(* Logix 5000 project; controller cal1615 1756-L62 rev 20.11; software revision 20.05; part 18 of 82 *)
(* tags used below, declared in another part *)
   FAULT : BOOL;   // Fault AFI
   HMI : BOOL;   // AFI HMI
   p01r09_pb_global_reset : BOOL;   // System Modes PB: Global Fault Reset
   p11_ai_exh_amps : REAL;   // Zone 1 Analog Input Exhaust Fan Amps
   p11_ai_exh_hz : REAL;   // Zone 1 Analog Input Exhaust Fan HZ
   p11_ai_exh_pct : REAL;   // Zone 1 Analog Input Exhaust Fan PCT
   p11_ai_exh_rpm : REAL;   // Zone 1 Analog Input Exhaust Fan RPM
   p11_ai_lfl : REAL;   // Zone 1 Analog Input Lower Flash Limit
   p11_ai_prs : REAL;   // Zone 1 Analog Input Pressure
   p11_ai_recirc_amps : REAL;   // Zone 1 Analog Input Recirc Fan Amps
   p11_ai_recirc_hz : REAL;   // Zone 1 Analog Input Supply Fan HZ
   p11_ai_recirc_pct : REAL;   // Zone 1 Analog Input Recirc Fan PCT
   p11_ai_recirc_rpm : REAL;   // Zone 1 Analog Input Recirc Fan RPM
   p11_ai_tc01 : REAL;   // Zone 1 Analog Input Control Thermocouple 1
   p11_ai_tc02 : REAL;   // Zone 1 Analog Input Control Thermocouple 2
   p11_ao_cv : REAL;   // Zone 1 Analog Output Control Valve
   p11_ao_exhaust_selected_speed : REAL;   // Zone 1 Analog Output Exhaust Fan VFD Selected Speed
   p11_ao_recirc_selected_speed : REAL;   // Zone 1 Analog Output Recirc Fan VFD Selected Speed
   p11_di_burner_auto : BOOL;   // Zone 1 Digital Input Burner Auto
   p11_di_burner_safeties_ok : BOOL;   // Zone 1 Digital Input Burner Safeties Ok
   p11_di_door_open : BOOL;   // Zone 1 Digital Input Access Door Open
   p11_di_exh : acs800_di_normal;   // Zone 1 Digital Inputs Exhaust Fan
   p11_di_exh_fan_mtr_ts : BOOL;   // Zone 1 Digital Input Exhaust Fan Motor Thermostat OK
   p11_di_exh_flow_ok : BOOL;   // Zone 1 Digital Input Exhaust Flow OK
   p11_di_flame_failure : BOOL;   // Zone 1 Digital Input Flame Failure
   p11_di_flame_on : BOOL;   // Zone 1 Digital Input Burner is On
   p11_di_fresh_air_clean : BOOL;   // Zone 1 Digital Input Fresh Air Filter Dirty
   p11_di_high_limit_temp_ok : BOOL;   // Zone 1 Digital Input High Limit Temperature OK
   p11_di_recirc : acs800_di_normal;   // Zone 1 Digital Inputs Recirc Fan
   p11_di_recirc_fan_mtr_ts : BOOL;   // Zone 1 Digital Input Recirc Fan Motor Thermostat OK
   p11_di_recirc_flow_ok : BOOL;   // Zone 1 Digital Input Recirc Flow OK
   p11_di_sp0 : BOOL;   // Zone 1 Digital Input Combustion Blower Pressure OK
   p11_di_sp00 : BOOL;   // Zone 1 Digital Input Recirculation Air Filter Dirty
   p11_di_tc01_bo : BOOL;   // Zone 1 Digital Input Control Thermocouple 1 Failure
   p11_di_tc02_bo : BOOL;   // Zone 1 Digital Input Control Thermocouple 2 Failure
   p11_di_zone_air_clean : BOOL;   // Zone 1 Digital Input Combustion Air Filter Dirty
   p11_dint_to_hmi : DINT[16];   // Zone 1 Temperature Control VFDs On
   p11_param_fast_to_soak : REAL;   // Zone 1 Parameter Fast to Soak Control
   p11_param_lfl_hhl : REAL;   // Zone 1 Parameter High High Lower Flash Limit
   p11_param_lfl_hl : REAL;   // Zone 1 Parameter High LFL Limit
   p11_param_pid1_ff : REAL;   // Zone 1 Parameter Fast PID Bias
   p11_param_pid1_kd : REAL;   // Zone 1 Parameter Fast PID Derivative Gain
   p11_param_pid1_ki : REAL;   // Zone 1 Parameter Fast PID Integral Gain
   p11_param_pid1_kp : REAL;   // Zone 1 Parameter Fast PID Proportional Gain
   p11_param_pid2_ff : REAL;   // Zone 1 Parameter Auto PID Bias
   p11_param_pid2_kd : REAL;   // Zone 1 Parameter Auto PID Derivative Gain
   p11_param_pid2_ki : REAL;   // Zone 1 Parameter Auto PID Integral Gain
   p11_param_pid2_kp : REAL;   // Zone 1 Parameter Auto PID Proportional Gain
   p11_param_shutdown_temp : REAL;   // Zone 1 Parameter Zone Shutdown Temperature
   p11_param_soak_to_fast : REAL;   // Zone 1 Parameter Soak to Fast Control
   p11_param_tc01_dev : REAL;   // Zone 1 Parameter Oven Temperature Deviation from Setpoint
   p11_param_tc01_hl : REAL;   // Zone 1 Parameter Process Air High Limit
   p11_param_tc01z : REAL;   // Zone 1 Parameter Process Temperature Zero Offset
   p11_param_tc02z : REAL;   // Zone 1 Parameter SupplyTemperature Zero Offset
   p11_param_zone_pressure : REAL;   // Zone 1 Parameter High Pressure LImit
   p11_real_to_hmi : REAL[112];   // Zone 1 Real to HMI
   p11r01 : routine;   // Zone 1 Main
   p11r05 : routine;   // Zone 1 Dint to HMI
   p11r05_exh_status : DINT;
   p11r05_recirc_status : DINT;
   p11r05_temp_ctrl_status : DINT;
   p11r05_timer_fault : TIMER[4];   // Zone 1 Dint to HMI Fault Delay
   p11r05_timer_warning : TIMER[4];   // Zone 1 Dint to HMI Warning Delay
   p11r06 : routine;   // Zone 1 Real to HMI
   p11r06_timer_fault : TIMER[4];   // Zone 1 Real to HMI Fault Delay
   p11r06_timer_warning : TIMER[4];   // Zone 1 Real to HMI Warning Delay
   p11r20_state : DINT;   // Zone 1 Temperature Control State
   p11r20_status : DINT;   // Zone 1 Temperature Control Sequence Status
   p11r30 : routine;   // Zone 1 Temperature Control
   p11r30_cv_man_sp : REAL;   // Zone 1 Temperature Control Manual Heat Control Valve Setpoint
   p11r30_permissive_run : BOOL;   // Zone 1 Temperature Control Run Permissive
   p11r30_pid_temp : PID;   // Zone 1 Temperature Control PID
   p11r30_pid_temp_pv : REAL;   // Zone 1 Temperature Control PID Temp Process Variable
   p11r30_pid_temp_sp : REAL;   // Zone 1 Temperature Control PID Temperature Control Setpoint
   p11r30_request_heat : BOOL;   // Zone 1 Temperature Control Request Heat
   p11r30_request_manual : BOOL;   // Zone 1 Temperature Control Request Manual Control
   p11r30_vfds_ready : BOOL;   // Zone 1 Temperature Control VFDs On
   p11r31 : routine;   // Zone 1 Exhaust VFD
   p11r31_request_auto_run : BOOL;   // Zone 1 Exhaust Fan Run Request
   p11r31_request_auto_stop : BOOL;   // Zone 1 Exhaust VFD Request Auto Stop
   p11r31_vfd_stopped : BOOL;   // Zone 1 Exhaust VFD VFD Stopped
   p11r32 : routine;   // Zone 1 Recirc VFD
   p11r32_request_auto_run : BOOL;   // Zone 1 Recirc Fan Run Request
   p11r32_request_auto_stop : BOOL;   // Zone 1 Recirc VFD Request Auto Stop
   p11r32_vfd_stopped : BOOL;   // Zone 1 Recirc VFD VFD Stopped
(* P11_Zone_1, continued *)

ROUTINE R05_Dint_to_HMI   (* ladder *)
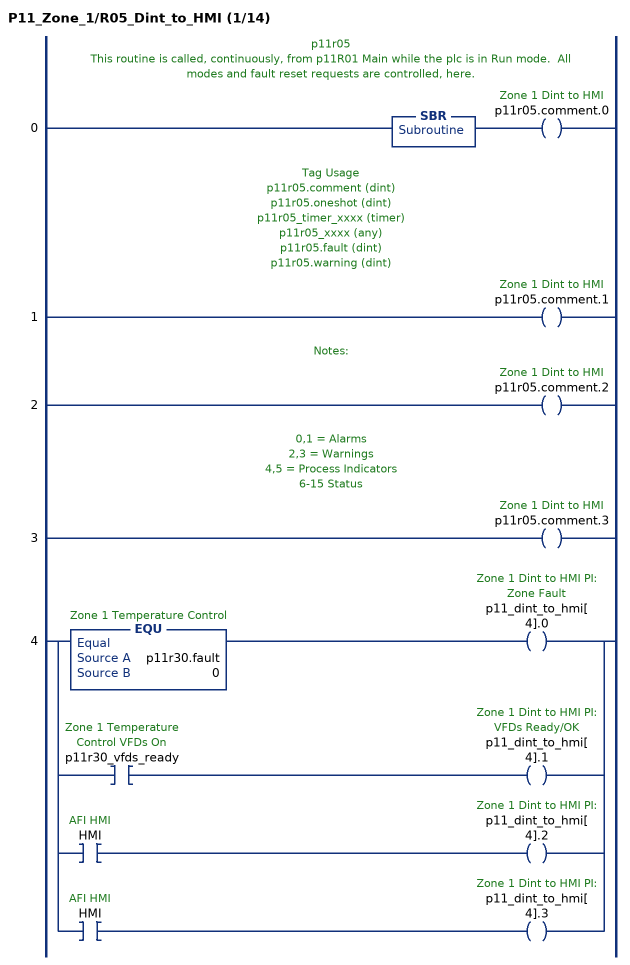
   // p11r05
   // This routine is called, continuously, from p11R01 Main while the plc is in Run mode.  All modes and fault reset requests are controlled, here.
   0: SBR()OTE(p11r05.comment.0);
   // Tag Usage
   // p11r05.comment (dint)
   // p11r05.oneshot (dint)
   // p11r05_timer_xxxx (timer)
   // p11r05_xxxx (any)
   // p11r05.fault (dint)
   // p11r05.warning (dint)
   1: OTE(p11r05.comment.1);
   // Notes:
   2: OTE(p11r05.comment.2);
   // 0,1 = Alarms
   // 2,3 = Warnings
   // 4,5 = Process Indicators
   // 6-15 Status
   3: OTE(p11r05.comment.3);
   4: [EQU(p11r30.fault,0) OTE(p11_dint_to_hmi[4].0) ,XIC(p11r30_vfds_ready) OTE(p11_dint_to_hmi[4].1) ,XIC(HMI) OTE(p11_dint_to_hmi[4].2) ,XIC(HMI) OTE(p11_dint_to_hmi[4].3) ];
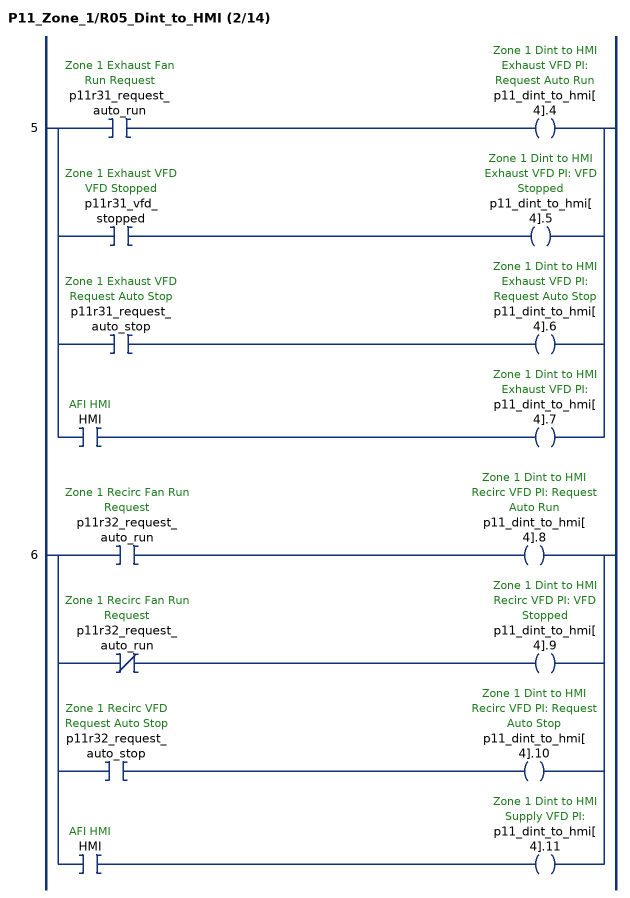
   5: [XIC(p11r31_request_auto_run) OTE(p11_dint_to_hmi[4].4) ,XIC(p11r31_vfd_stopped) OTE(p11_dint_to_hmi[4].5) ,XIC(p11r31_request_auto_stop) OTE(p11_dint_to_hmi[4].6) ,XIC(HMI) OTE(p11_dint_to_hmi[4].7) ];
   6: [XIC(p11r32_request_auto_run) OTE(p11_dint_to_hmi[4].8) ,XIO(p11r32_request_auto_run) OTE(p11_dint_to_hmi[4].9) ,XIC(p11r32_request_auto_stop) OTE(p11_dint_to_hmi[4].10) ,XIC(HMI) OTE(p11_dint_to_hmi[4].11) ];
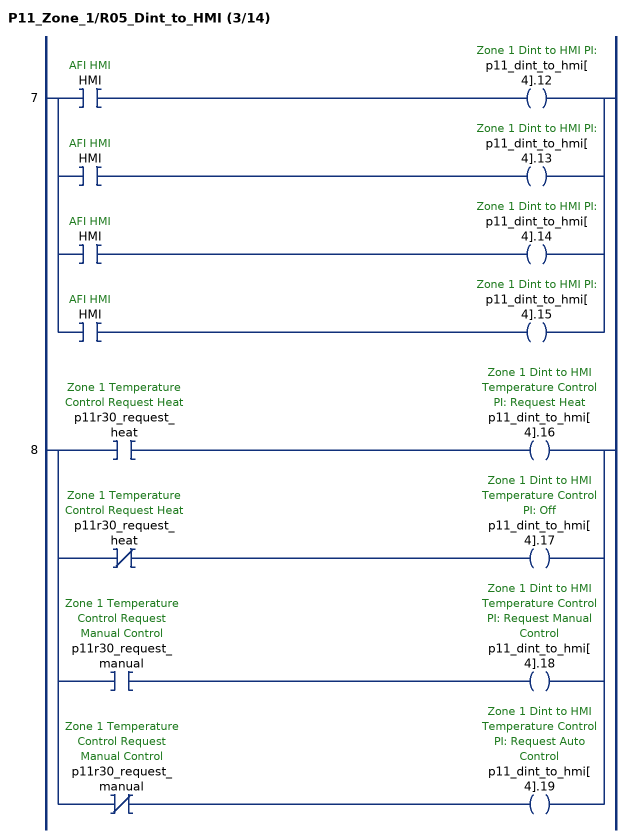
   7: [XIC(HMI) OTE(p11_dint_to_hmi[4].12) ,XIC(HMI) OTE(p11_dint_to_hmi[4].13) ,XIC(HMI) OTE(p11_dint_to_hmi[4].14) ,XIC(HMI) OTE(p11_dint_to_hmi[4].15) ];
   8: [XIC(p11r30_request_heat) OTE(p11_dint_to_hmi[4].16) ,XIO(p11r30_request_heat) OTE(p11_dint_to_hmi[4].17) ,XIC(p11r30_request_manual) OTE(p11_dint_to_hmi[4].18) ,XIO(p11r30_request_manual) OTE(p11_dint_to_hmi[4].19) ];
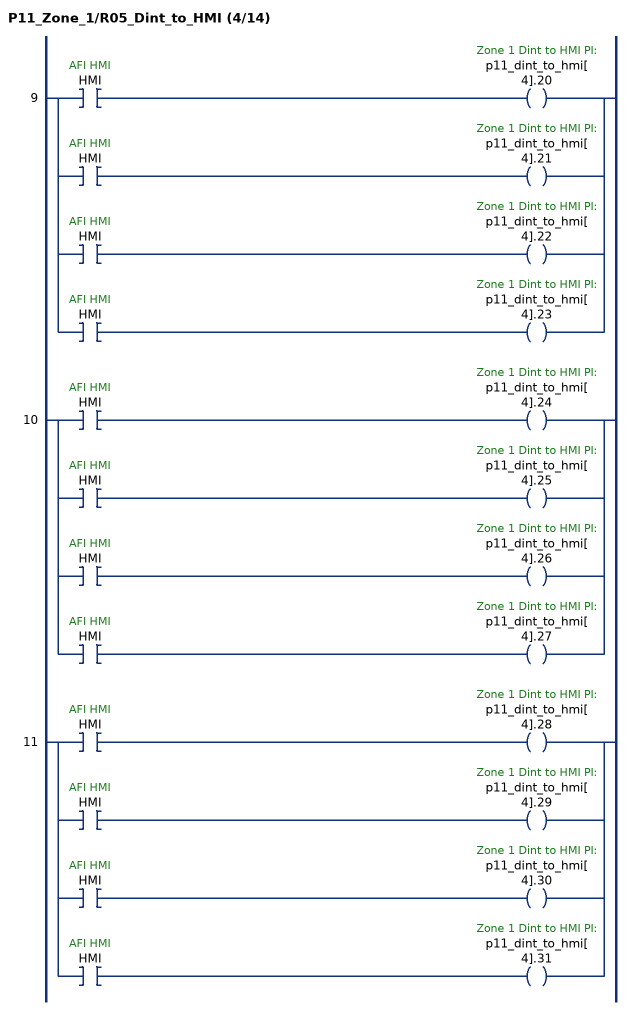
   9: [XIC(HMI) OTE(p11_dint_to_hmi[4].20) ,XIC(HMI) OTE(p11_dint_to_hmi[4].21) ,XIC(HMI) OTE(p11_dint_to_hmi[4].22) ,XIC(HMI) OTE(p11_dint_to_hmi[4].23) ];
   10: [XIC(HMI) OTE(p11_dint_to_hmi[4].24) ,XIC(HMI) OTE(p11_dint_to_hmi[4].25) ,XIC(HMI) OTE(p11_dint_to_hmi[4].26) ,XIC(HMI) OTE(p11_dint_to_hmi[4].27) ];
   11: [XIC(HMI) OTE(p11_dint_to_hmi[4].28) ,XIC(HMI) OTE(p11_dint_to_hmi[4].29) ,XIC(HMI) OTE(p11_dint_to_hmi[4].30) ,XIC(HMI) OTE(p11_dint_to_hmi[4].31) ];
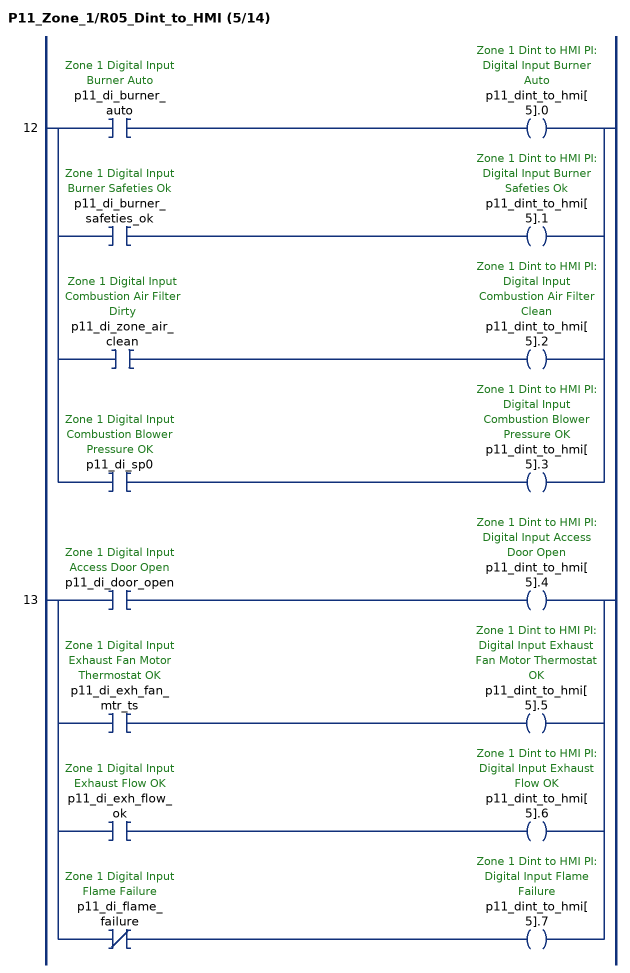
   12: [XIC(p11_di_burner_auto) OTE(p11_dint_to_hmi[5].0) ,XIC(p11_di_burner_safeties_ok) OTE(p11_dint_to_hmi[5].1) ,XIC(p11_di_zone_air_clean) OTE(p11_dint_to_hmi[5].2) ,XIC(p11_di_sp0) OTE(p11_dint_to_hmi[5].3) ];
   13: [XIC(p11_di_door_open) OTE(p11_dint_to_hmi[5].4) ,XIC(p11_di_exh_fan_mtr_ts) OTE(p11_dint_to_hmi[5].5) ,XIC(p11_di_exh_flow_ok) OTE(p11_dint_to_hmi[5].6) ,XIO(p11_di_flame_failure) OTE(p11_dint_to_hmi[5].7) ];
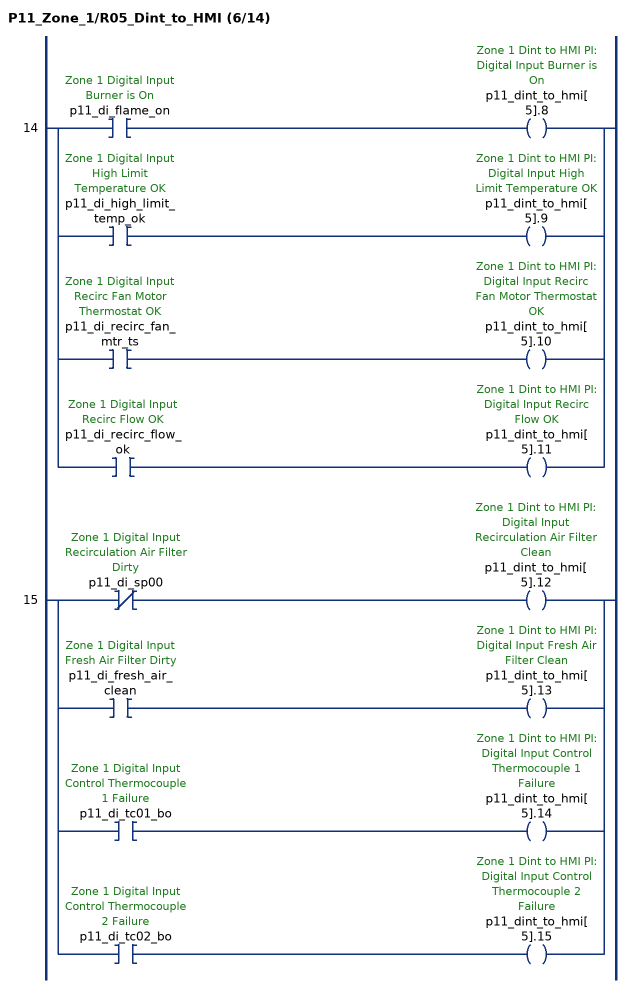
   14: [XIC(p11_di_flame_on) OTE(p11_dint_to_hmi[5].8) ,XIC(p11_di_high_limit_temp_ok) OTE(p11_dint_to_hmi[5].9) ,XIC(p11_di_recirc_fan_mtr_ts) OTE(p11_dint_to_hmi[5].10) ,XIC(p11_di_recirc_flow_ok) OTE(p11_dint_to_hmi[5].11) ];
   15: [XIO(p11_di_sp00) OTE(p11_dint_to_hmi[5].12) ,XIC(p11_di_fresh_air_clean) OTE(p11_dint_to_hmi[5].13) ,XIC(p11_di_tc01_bo) OTE(p11_dint_to_hmi[5].14) ,XIC(p11_di_tc02_bo) OTE(p11_dint_to_hmi[5].15) ];
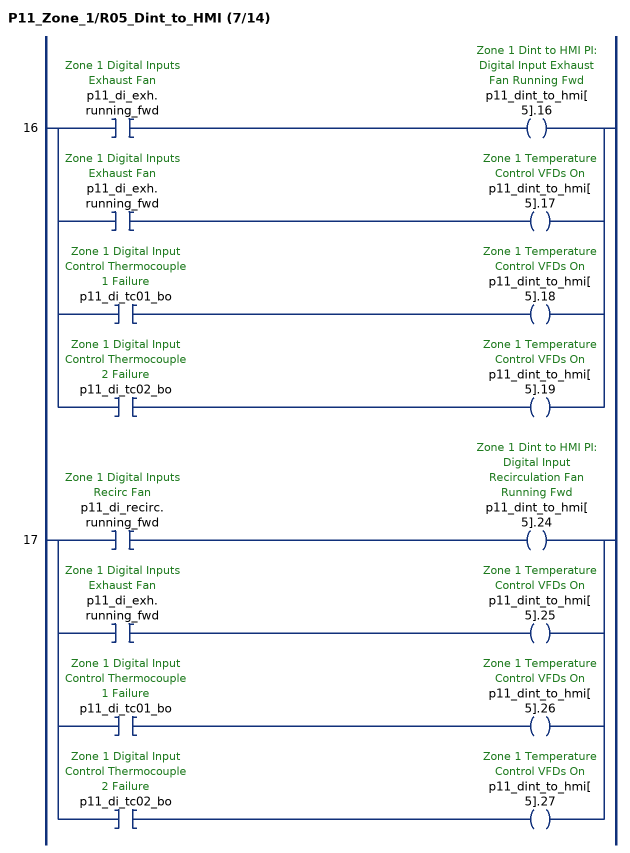
   16: [XIC(p11_di_exh.running_fwd) OTE(p11_dint_to_hmi[5].16) ,XIC(p11_di_exh.running_fwd) OTE(p11_dint_to_hmi[5].17) ,XIC(p11_di_tc01_bo) OTE(p11_dint_to_hmi[5].18) ,XIC(p11_di_tc02_bo) OTE(p11_dint_to_hmi[5].19) ];
   17: [XIC(p11_di_recirc.running_fwd) OTE(p11_dint_to_hmi[5].24) ,XIC(p11_di_exh.running_fwd) OTE(p11_dint_to_hmi[5].25) ,XIC(p11_di_tc01_bo) OTE(p11_dint_to_hmi[5].26) ,XIC(p11_di_tc02_bo) OTE(p11_dint_to_hmi[5].27) ];
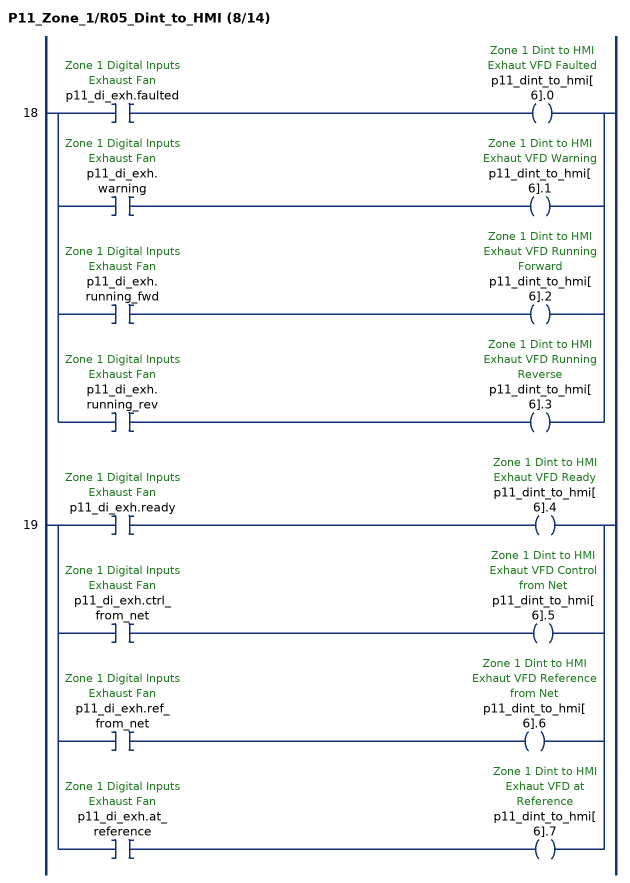
   18: [XIC(p11_di_exh.faulted) OTE(p11_dint_to_hmi[6].0) ,XIC(p11_di_exh.warning) OTE(p11_dint_to_hmi[6].1) ,XIC(p11_di_exh.running_fwd) OTE(p11_dint_to_hmi[6].2) ,XIC(p11_di_exh.running_rev) OTE(p11_dint_to_hmi[6].3) ];
   19: [XIC(p11_di_exh.ready) OTE(p11_dint_to_hmi[6].4) ,XIC(p11_di_exh.ctrl_from_net) OTE(p11_dint_to_hmi[6].5) ,XIC(p11_di_exh.ref_from_net) OTE(p11_dint_to_hmi[6].6) ,XIC(p11_di_exh.at_reference) OTE(p11_dint_to_hmi[6].7) ];
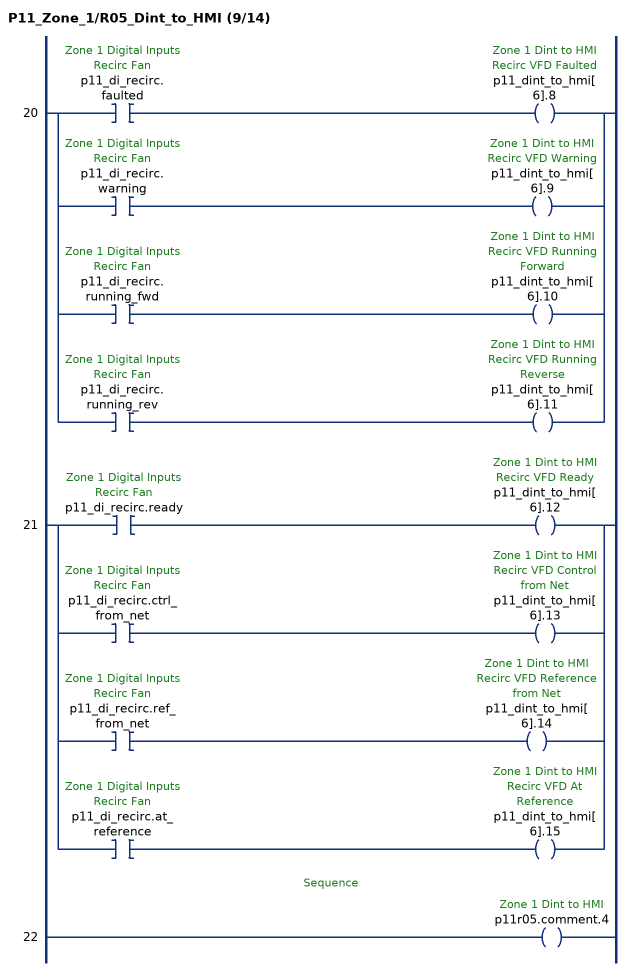
   20: [XIC(p11_di_recirc.faulted) OTE(p11_dint_to_hmi[6].8) ,XIC(p11_di_recirc.warning) OTE(p11_dint_to_hmi[6].9) ,XIC(p11_di_recirc.running_fwd) OTE(p11_dint_to_hmi[6].10) ,XIC(p11_di_recirc.running_rev) OTE(p11_dint_to_hmi[6].11) ];
   21: [XIC(p11_di_recirc.ready) OTE(p11_dint_to_hmi[6].12) ,XIC(p11_di_recirc.ctrl_from_net) OTE(p11_dint_to_hmi[6].13) ,XIC(p11_di_recirc.ref_from_net) OTE(p11_dint_to_hmi[6].14) ,XIC(p11_di_recirc.at_reference) OTE(p11_dint_to_hmi[6].15) ];
   // Sequence
   22: OTE(p11r05.comment.4);
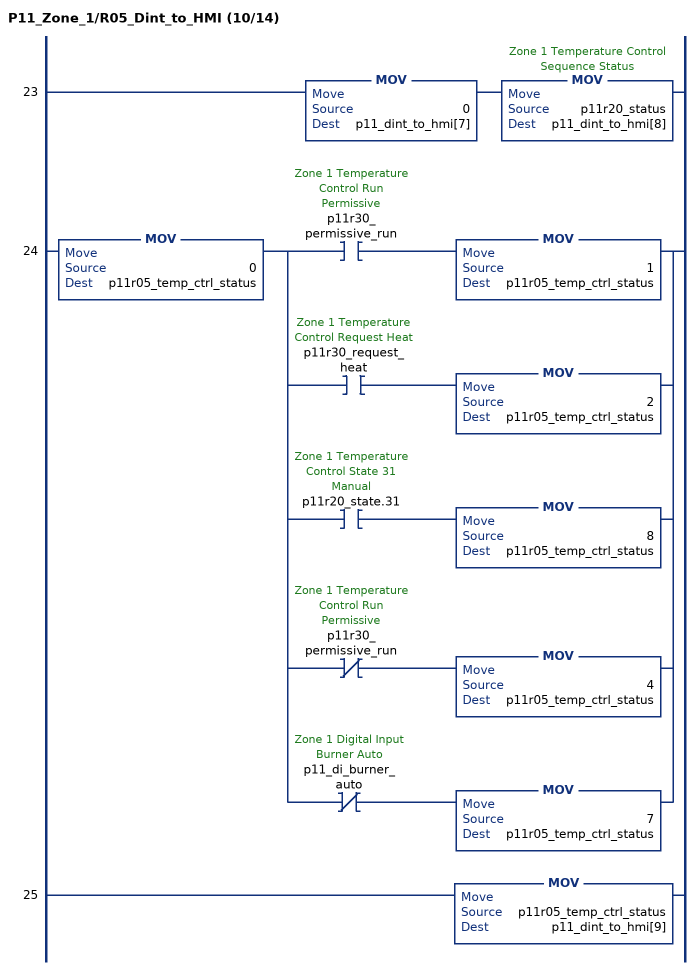
   23: MOV(0,p11_dint_to_hmi[7])MOV(p11r20_status,p11_dint_to_hmi[8]);
   24: MOV(0,p11r05_temp_ctrl_status)[XIC(p11r30_permissive_run) MOV(1,p11r05_temp_ctrl_status) ,XIC(p11r30_request_heat) MOV(2,p11r05_temp_ctrl_status) ,XIC(p11r20_state.31) MOV(8,p11r05_temp_ctrl_status) ,XIO(p11r30_permissive_run) MOV(4,p11r05_temp_ctrl_status) ,XIO(p11_di_burner_auto) MOV(7,p11r05_temp_ctrl_status) ];
   25: MOV(p11r05_temp_ctrl_status,p11_dint_to_hmi[9]);
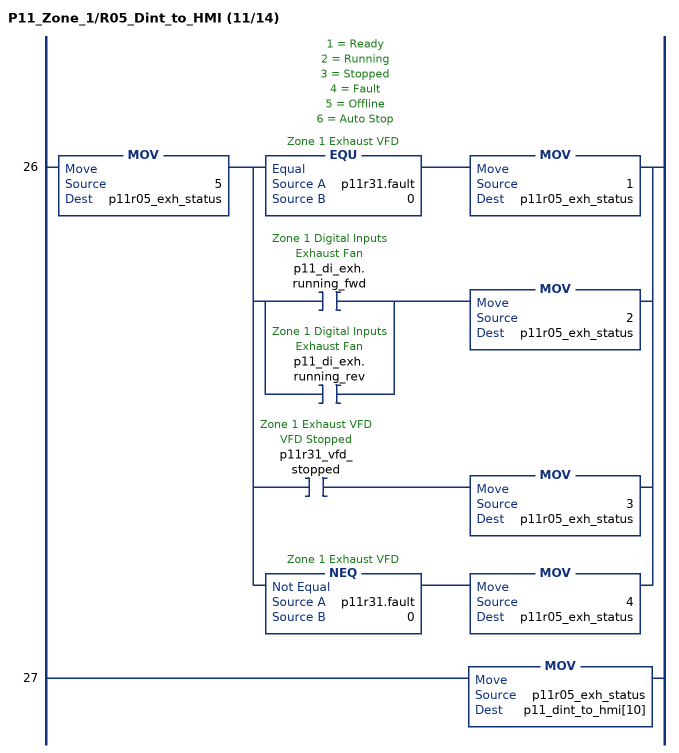
   // 1 = Ready
   // 2 = Running
   // 3 = Stopped
   // 4 = Fault
   // 5 = Offline
   // 6 = Auto Stop
   26: MOV(5,p11r05_exh_status)[EQU(p11r31.fault,0) MOV(1,p11r05_exh_status) ,[XIC(p11_di_exh.running_fwd) ,XIC(p11_di_exh.running_rev) ] MOV(2,p11r05_exh_status) ,XIC(p11r31_vfd_stopped) MOV(3,p11r05_exh_status) ,NEQ(p11r31.fault,0) MOV(4,p11r05_exh_status) ];
   27: MOV(p11r05_exh_status,p11_dint_to_hmi[10]);
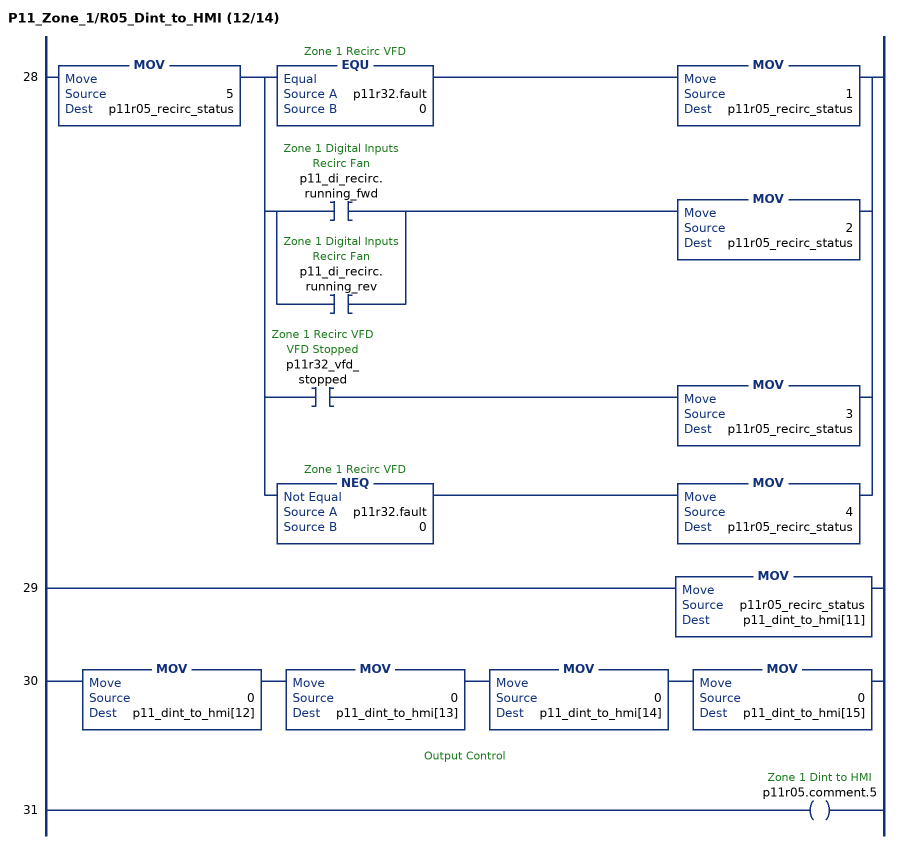
   28: MOV(5,p11r05_recirc_status)[EQU(p11r32.fault,0) MOV(1,p11r05_recirc_status) ,[XIC(p11_di_recirc.running_fwd) ,XIC(p11_di_recirc.running_rev) ] MOV(2,p11r05_recirc_status) ,XIC(p11r32_vfd_stopped) MOV(3,p11r05_recirc_status) ,NEQ(p11r32.fault,0) MOV(4,p11r05_recirc_status) ];
   29: MOV(p11r05_recirc_status,p11_dint_to_hmi[11]);
   30: MOV(0,p11_dint_to_hmi[12])MOV(0,p11_dint_to_hmi[13])MOV(0,p11_dint_to_hmi[14])MOV(0,p11_dint_to_hmi[15]);
   // Output Control
   31: OTE(p11r05.comment.5);
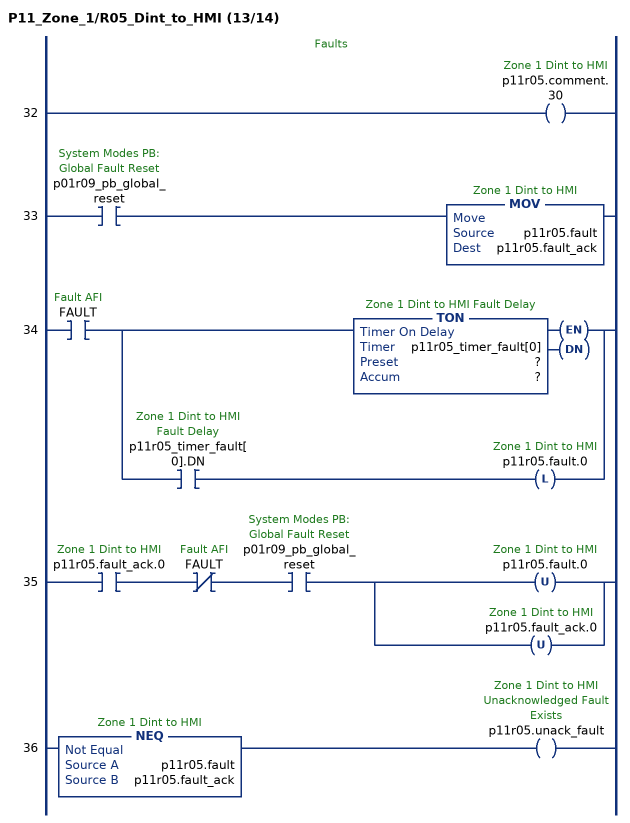
   // Faults
   32: OTE(p11r05.comment.30);
   33: XIC(p01r09_pb_global_reset)MOV(p11r05.fault,p11r05.fault_ack);
   34: XIC(FAULT)[TON(p11r05_timer_fault[0],?,?) ,XIC(p11r05_timer_fault[0].DN) OTL(p11r05.fault.0) ];
   35: XIC(p11r05.fault_ack.0)XIO(FAULT)XIC(p01r09_pb_global_reset)[OTU(p11r05.fault.0) ,OTU(p11r05.fault_ack.0) ];
   36: NEQ(p11r05.fault,p11r05.fault_ack)OTE(p11r05.unack_fault);
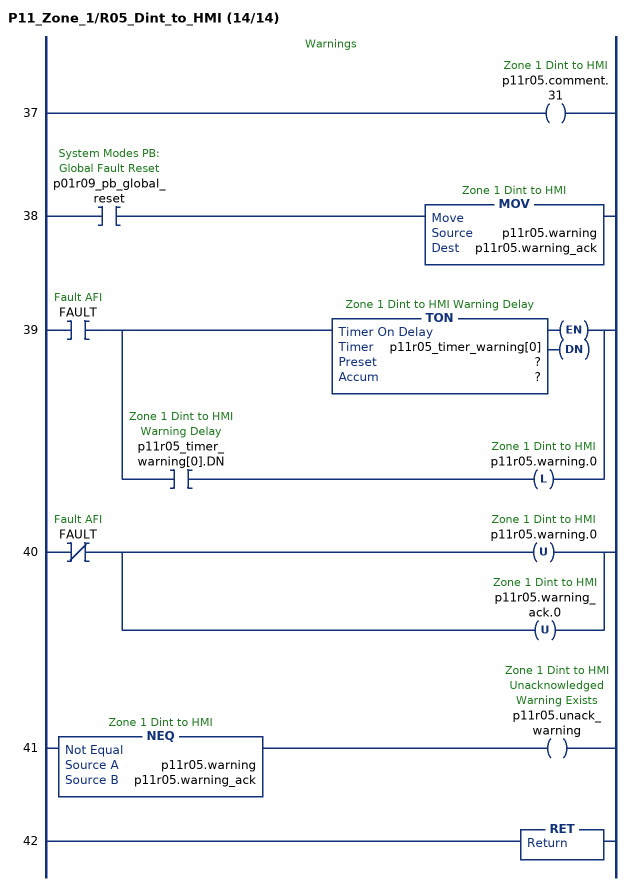
   // Warnings
   37: OTE(p11r05.comment.31);
   38: XIC(p01r09_pb_global_reset)MOV(p11r05.warning,p11r05.warning_ack);
   39: XIC(FAULT)[TON(p11r05_timer_warning[0],?,?) ,XIC(p11r05_timer_warning[0].DN) OTL(p11r05.warning.0) ];
   40: XIO(FAULT)[OTU(p11r05.warning.0) ,OTU(p11r05.warning_ack.0) ];
   41: NEQ(p11r05.warning,p11r05.warning_ack)OTE(p11r05.unack_warning);
   42: RET();
END_ROUTINE

ROUTINE R06_Real_to_HMI   (* ladder *)
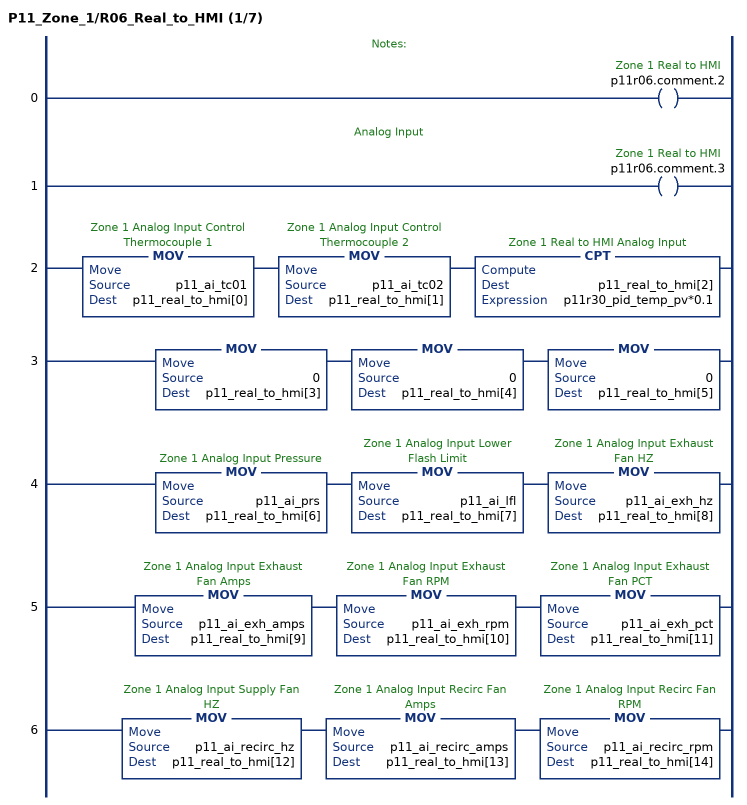
   // Notes:
   0: OTE(p11r06.comment.2);
   // Analog Input
   1: OTE(p11r06.comment.3);
   2: MOV(p11_ai_tc01,p11_real_to_hmi[0])MOV(p11_ai_tc02,p11_real_to_hmi[1])CPT(p11_real_to_hmi[2],p11r30_pid_temp_pv*0.1);
   3: MOV(0,p11_real_to_hmi[3])MOV(0,p11_real_to_hmi[4])MOV(0,p11_real_to_hmi[5]);
   4: MOV(p11_ai_prs,p11_real_to_hmi[6])MOV(p11_ai_lfl,p11_real_to_hmi[7])MOV(p11_ai_exh_hz,p11_real_to_hmi[8]);
   5: MOV(p11_ai_exh_amps,p11_real_to_hmi[9])MOV(p11_ai_exh_rpm,p11_real_to_hmi[10])MOV(p11_ai_exh_pct,p11_real_to_hmi[11]);
   6: MOV(p11_ai_recirc_hz,p11_real_to_hmi[12])MOV(p11_ai_recirc_amps,p11_real_to_hmi[13])MOV(p11_ai_recirc_rpm,p11_real_to_hmi[14]);
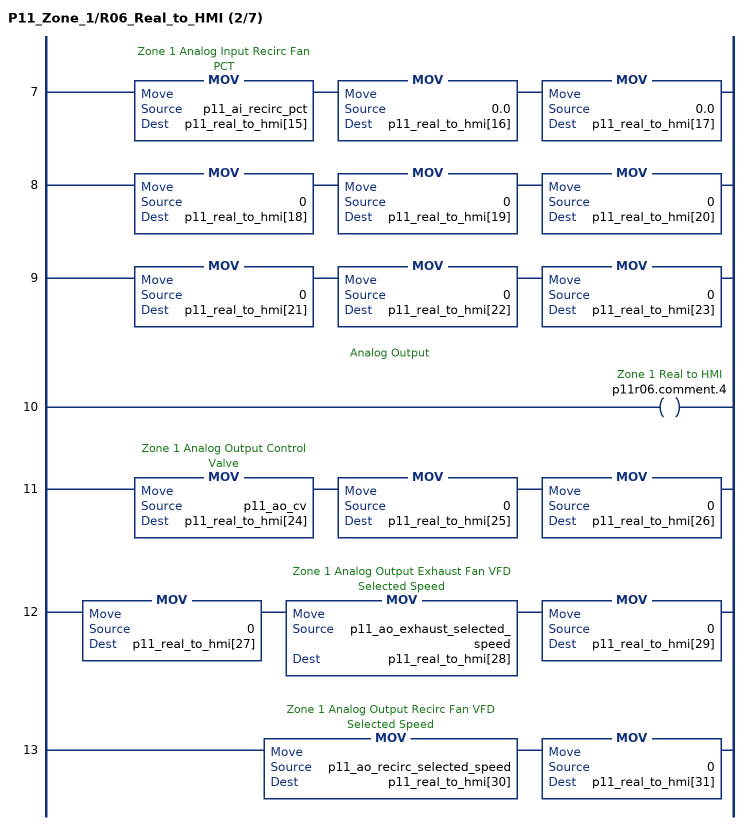
   7: MOV(p11_ai_recirc_pct,p11_real_to_hmi[15])MOV(0.0,p11_real_to_hmi[16])MOV(0.0,p11_real_to_hmi[17]);
   8: MOV(0,p11_real_to_hmi[18])MOV(0,p11_real_to_hmi[19])MOV(0,p11_real_to_hmi[20]);
   9: MOV(0,p11_real_to_hmi[21])MOV(0,p11_real_to_hmi[22])MOV(0,p11_real_to_hmi[23]);
   // Analog Output
   10: OTE(p11r06.comment.4);
   11: MOV(p11_ao_cv,p11_real_to_hmi[24])MOV(0,p11_real_to_hmi[25])MOV(0,p11_real_to_hmi[26]);
   12: MOV(0,p11_real_to_hmi[27])MOV(p11_ao_exhaust_selected_speed,p11_real_to_hmi[28])MOV(0,p11_real_to_hmi[29]);
   13: MOV(p11_ao_recirc_selected_speed,p11_real_to_hmi[30])MOV(0,p11_real_to_hmi[31]);
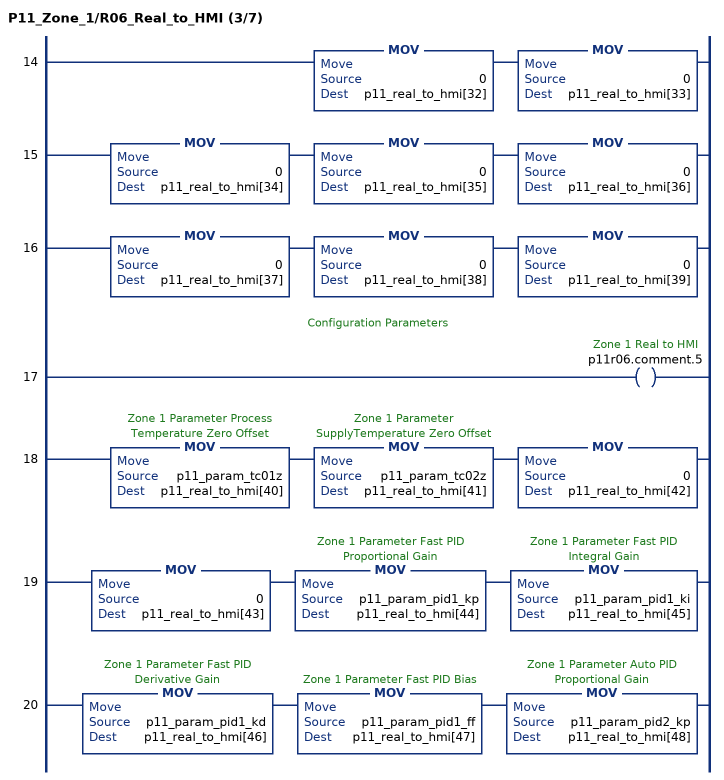
   14: MOV(0,p11_real_to_hmi[32])MOV(0,p11_real_to_hmi[33]);
   15: MOV(0,p11_real_to_hmi[34])MOV(0,p11_real_to_hmi[35])MOV(0,p11_real_to_hmi[36]);
   16: MOV(0,p11_real_to_hmi[37])MOV(0,p11_real_to_hmi[38])MOV(0,p11_real_to_hmi[39]);
   // Configuration Parameters
   17: OTE(p11r06.comment.5);
   18: MOV(p11_param_tc01z,p11_real_to_hmi[40])MOV(p11_param_tc02z,p11_real_to_hmi[41])MOV(0,p11_real_to_hmi[42]);
   19: MOV(0,p11_real_to_hmi[43])MOV(p11_param_pid1_kp,p11_real_to_hmi[44])MOV(p11_param_pid1_ki,p11_real_to_hmi[45]);
   20: MOV(p11_param_pid1_kd,p11_real_to_hmi[46])MOV(p11_param_pid1_ff,p11_real_to_hmi[47])MOV(p11_param_pid2_kp,p11_real_to_hmi[48]);
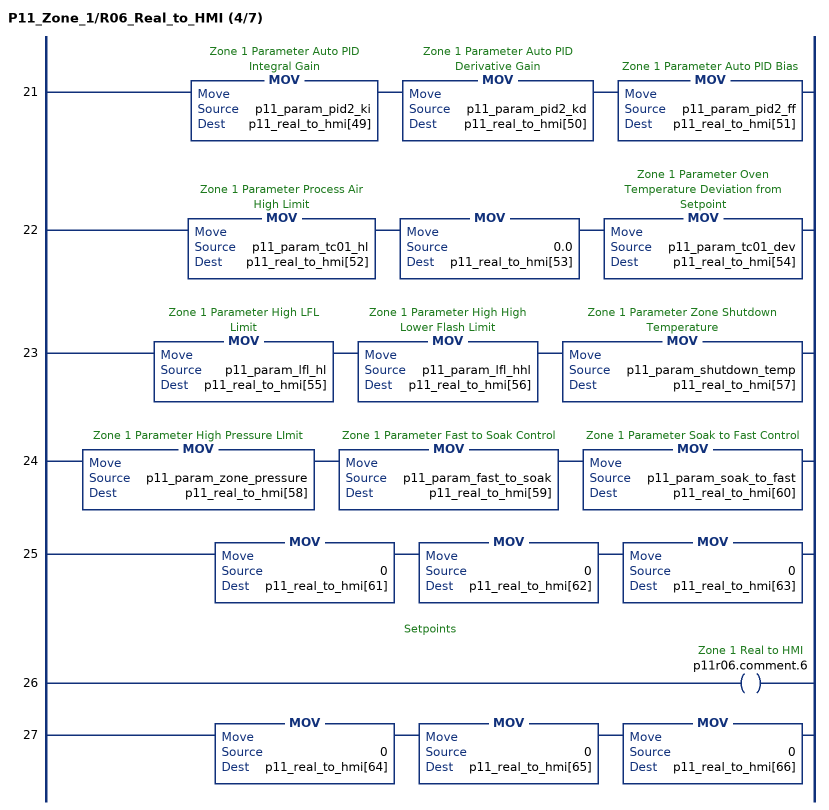
   21: MOV(p11_param_pid2_ki,p11_real_to_hmi[49])MOV(p11_param_pid2_kd,p11_real_to_hmi[50])MOV(p11_param_pid2_ff,p11_real_to_hmi[51]);
   22: MOV(p11_param_tc01_hl,p11_real_to_hmi[52])MOV(0.0,p11_real_to_hmi[53])MOV(p11_param_tc01_dev,p11_real_to_hmi[54]);
   23: MOV(p11_param_lfl_hl,p11_real_to_hmi[55])MOV(p11_param_lfl_hhl,p11_real_to_hmi[56])MOV(p11_param_shutdown_temp,p11_real_to_hmi[57]);
   24: MOV(p11_param_zone_pressure,p11_real_to_hmi[58])MOV(p11_param_fast_to_soak,p11_real_to_hmi[59])MOV(p11_param_soak_to_fast,p11_real_to_hmi[60]);
   25: MOV(0,p11_real_to_hmi[61])MOV(0,p11_real_to_hmi[62])MOV(0,p11_real_to_hmi[63]);
   // Setpoints
   26: OTE(p11r06.comment.6);
   27: MOV(0,p11_real_to_hmi[64])MOV(0,p11_real_to_hmi[65])MOV(0,p11_real_to_hmi[66]);
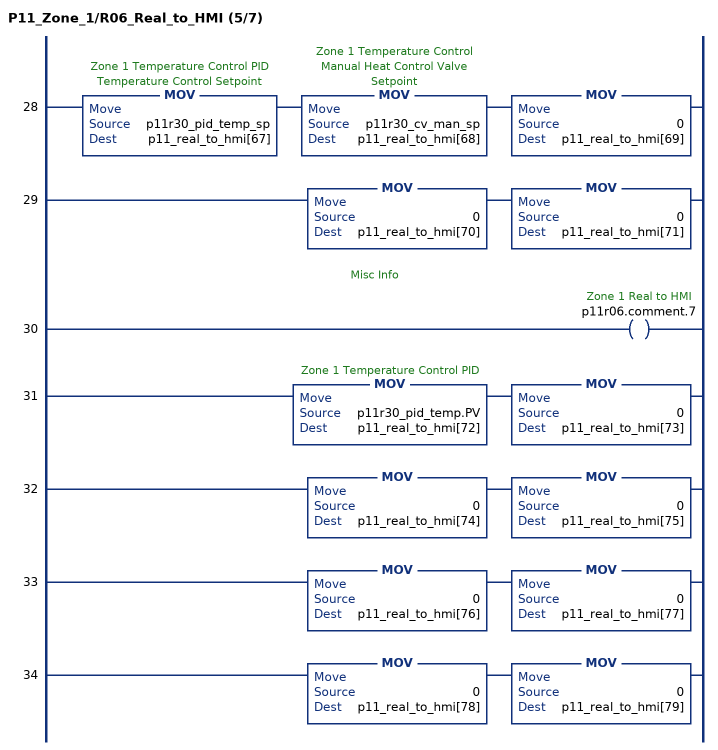
   28: MOV(p11r30_pid_temp_sp,p11_real_to_hmi[67])MOV(p11r30_cv_man_sp,p11_real_to_hmi[68])MOV(0,p11_real_to_hmi[69]);
   29: MOV(0,p11_real_to_hmi[70])MOV(0,p11_real_to_hmi[71]);
   // Misc Info
   30: OTE(p11r06.comment.7);
   31: MOV(p11r30_pid_temp.PV,p11_real_to_hmi[72])MOV(0,p11_real_to_hmi[73]);
   32: MOV(0,p11_real_to_hmi[74])MOV(0,p11_real_to_hmi[75]);
   33: MOV(0,p11_real_to_hmi[76])MOV(0,p11_real_to_hmi[77]);
   34: MOV(0,p11_real_to_hmi[78])MOV(0,p11_real_to_hmi[79]);
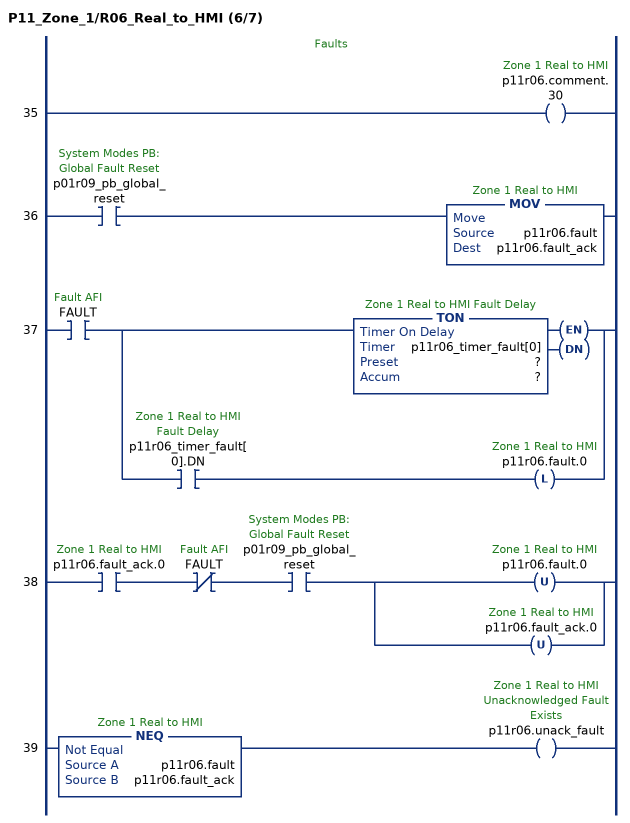
   // Faults
   35: OTE(p11r06.comment.30);
   36: XIC(p01r09_pb_global_reset)MOV(p11r06.fault,p11r06.fault_ack);
   37: XIC(FAULT)[TON(p11r06_timer_fault[0],?,?) ,XIC(p11r06_timer_fault[0].DN) OTL(p11r06.fault.0) ];
   38: XIC(p11r06.fault_ack.0)XIO(FAULT)XIC(p01r09_pb_global_reset)[OTU(p11r06.fault.0) ,OTU(p11r06.fault_ack.0) ];
   39: NEQ(p11r06.fault,p11r06.fault_ack)OTE(p11r06.unack_fault);
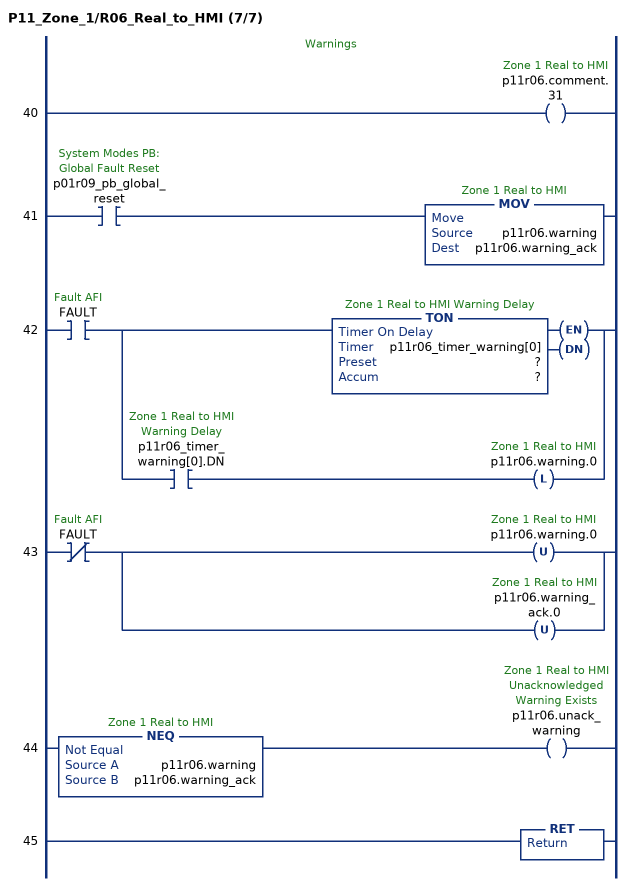
   // Warnings
   40: OTE(p11r06.comment.31);
   41: XIC(p01r09_pb_global_reset)MOV(p11r06.warning,p11r06.warning_ack);
   42: XIC(FAULT)[TON(p11r06_timer_warning[0],?,?) ,XIC(p11r06_timer_warning[0].DN) OTL(p11r06.warning.0) ];
   43: XIO(FAULT)[OTU(p11r06.warning.0) ,OTU(p11r06.warning_ack.0) ];
   44: NEQ(p11r06.warning,p11r06.warning_ack)OTE(p11r06.unack_warning);
   45: RET();
END_ROUTINE
